ABB RobotStudio station: parte 2 - Lisandro y Camila.rspag

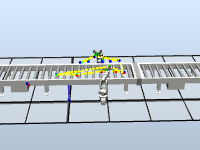
--- station ---
Station PARCIAL_FINAL_20 (saved by RobotStudio 6.8.8307.1040)
Controller IRB_120_3kg_0.58m_izqueirdo, task T_ROB1: task frame (RAPID world) sits at (1975.54, -890.46, 0) mm, rotated rx 0 ry 0 rz 180 deg in the station
Controller IRB_120_3kg_0.58m, task T_ROB1: task frame (RAPID world) sits at (-16.49, -890.46, 0) mm in the station
Controller IRB_120_3kg_0.58m
  mechanical unit ROB_1: IRB120_derecho, 6 joints, base frame (0, 0, 0) mm
Controller IRB_120_3kg_0.58m_izqueirdo
  mechanical unit ROB_1: IRB120_izquierdo, 6 joints, base frame (0, 0, 0) mm
Layout (positions relative to the parent item):
  - IRB120_derecho [mechanism] at (-16.49, -890.46, 0) mm; joint values [-0.3384, 0.2785, -0.49, -0.1645, -0.0408, 0.5646] (rad or m)
      links: Base, Link1, Link2, Link3, Link4, Link5, Link6
  - MyTool_derecho [mechanism] at (384.12, -1030.96, 699.37) mm, rotated rx 56.47 ry 63.2 rz 40.4 deg
      TCP MyTool at (31.79, 0, 229.64) mm, rotated rx 0 ry 38 rz 0 deg
      links: SpintecTool
  - SmartComponent_1 [smart component]
      signals: DI INICIO, DO DONE_1, DO WAIT_ROBOT, DI WAIT_ROBOT_1
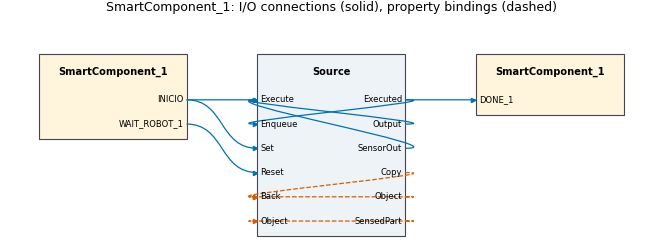
      connections:
        SmartComponent_1.INICIO -> Source.Execute
        Source.Executed -> Queue.Enqueue
        LogicSRLatch_2.Output -> LinearMover.Execute
        SmartComponent_1.INICIO -> LogicSRLatch_2.Set
        LineSensor.SensorOut -> Sink.Execute
        Sink.Executed -> SmartComponent_1.DONE_1
        SmartComponent_1.WAIT_ROBOT_1 -> LogicSRLatch_2.Reset
        Source.Copy => Queue.Back
        LinearMover.Object => Queue.Back
        LineSensor.SensedPart => Sink.Object
    - 950_4000_h2 [part] at (481.84, -1943.26, 0) mm, rotated rx 0 ry 0 rz -90 deg
    - 950_4000 [part] at (481.84, 2303.05, 0) mm, rotated rx 0 ry 0 rz -90 deg
  - LineSensor_3 [smart component, from Components\LineSensor.rslib] at (0, 0, 82.21) mm
      properties: Start=[0.481837 -1.468577 0.417790711533662]; End=[1.391837 -1.454228 0.417790711533662]; Radius=0; SensedPart=(none); SensedPoint=[1.1188828125 -1.45853198242187 0.5]
    - _sensorPart_ [part]
  - LinearMover_5 [smart component, from Components\LinearMover.rslib]
      properties: Object=(none); Direction=[0 -5 0]; Speed=0.45; Reference=Global; ReferenceObject=(none)
  - LogicSRLatch_3 [smart component, from Components\LogicSRLatch.rslib]
  - carro v10_9 [part] at (845.35, 1324.55, 563.17) mm, rotated rx 90 ry 0 rz 90 deg
  - Queue [smart component, from Components\Queue.rslib]
      properties: Back=(none); Front=(none); Queue={2e9f6991-8765-46e1-b9d2-2ffc72d677af};{ae45a596-02e8-4e52-9286-656ae225cacd};{e6612efd-c0eb-488b-85f8-b7f4c3102223};{41649e3c-b784-4099-a2b6-5bbce63e6931};{7cccd143-9200-41c9-9571-56f89e3b47af};{9ae8a6fd-c274-4031-a548-9f3ef3f36b3a};{8e4b5e29-5d32-45ba-96b5-431f4aa4aeb4};{b12dc332-1d97-4a47-8d88-8e0bee83711f};{b06eb078-9d15-4dac-a639-ca4a5d045752};{36dd95e1-a525-41dc-89b9-a063a131a275};{90e40d64-8709-426d-9514-00f99289b4fd};{8238a00f-e375-4470-8a06-12bd71f22f04};{9cebabc8-3cf8-4b9a-aff2-1a40ba7d75c4};{e08df943-d758-42c3-b96e-c5a5a5535acf};{779e000a-15d6-42ef-9bae-f04b49e1bf69};{19063376-c3c8-401e-bc56-325a5b5330d4};{6fb3a925-9c96-444a-9cf6-2b48ab2bb77b};{b99dccf3-a9df-44c4-8768-e74e9a577921};{d042e8a6-24ab-4afd-8b08-62ef72f8d954};{469562c5-238e-4f1a-8a6a-e243ac061d49};{98599022-264f-40f7-abfe-657128622a59};{93bca168-39dd-414b-b794-00b031783849};{70e5a896-b097-490d-8be8-28998b22b420};{5813b6a1-ddc2-47c4-ac52-396df1c672e9};{180ec9fe-a73e-4834-8773-2bd90c542f4d};{68088890-b0b0-44d4-a72b-623dbc1f9591};{e385e6d6-b519-43fc-8129-9058077c405e};{fb7d959f-a590-4f16-a74b-a7969766d88b};{d415407e-bbc8-41df-8733-1a202f62ccfb};{3bfff912-d452-4fed-8fb6-201deedca72a};{e2d4b341-78bb-44fa-a800-ceced0670a4f};{baedb794-50eb-4695-9b41-42448fe955b1};{10d86464-9892-4255-8e29-7578ef2925c7};{514a4022-64fc-47d2-bc88-f3ff3a7435df};{87afceb3-19d2-40d5-b81b-794861be6da1};{30505d37-60bd-4412-8ca7-5a9feadde122};{d50750b3-7fed-419f-9bb7-134f78306727};{72818c27-da5f-4208-8d82-50bde2b66c7d}; NumberOfObjects=1
  - Sink [smart component, from Components\Sink.rslib]
      properties: Object=(none)
  - Source [smart component, from Components\Source.rslib]
      properties: Source=carro v10_9; Copy=(none); Parent=(none); Position=[0.84535 1.32455 0.56317]; Orientation=[1.5707963267949 0 1.5707963267949]; Transient=false; PhysicsBehavior=2
  - LinearMover_6 [smart component, from Components\LinearMover.rslib]
      properties: Object=(none); Direction=[0 -6 0]; Speed=0.45; Reference=Global; ReferenceObject=(none)
  - LogicSRLatch_4 [smart component, from Components\LogicSRLatch.rslib]
  - LineSensor_4 [smart component, from Components\LineSensor.rslib]
      properties: Start=[0.481837 -3.897492 0.5]; End=[1.391837 -3.903973 0.5]; Radius=0; SensedPart=(none); SensedPoint=[0 0 0]
    - _sensorPart_ [part]
  - MyTool_izquierdo [mechanism] at (1574.94, -749.96, 699.37) mm, rotated rx 56.47 ry 63.2 rz -139.6 deg
      TCP MyTool at (31.79, 0, 229.64) mm, rotated rx 0 ry 38 rz 0 deg
      links: SpintecTool
  - IRB120_izquierdo [mechanism] at (1975.54, -890.46, 0) mm, rotated rx 0 ry 0 rz 180 deg; joint values [-0.3384, 0.2785, -0.49, -0.1645, -0.0408, 0.5645] (rad or m)
      links: Base, Link1, Link2, Link3, Link4, Link5, Link6
Attachment: MyTool_derecho is attached to IRB120_derecho / Link6
Attachment: MyTool_izquierdo is attached to IRB120_izquierdo / Link6
Station signals: DI STAR_JOB, DI RESET_CARRITO, DO END
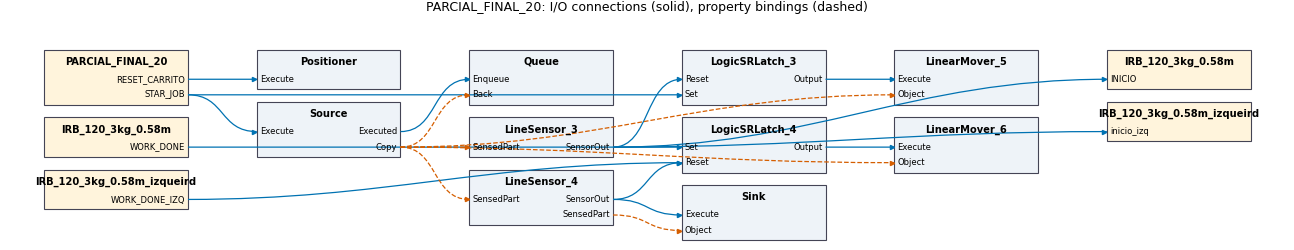
Station logic (signal -> signal, property => property):
  LineSensor_3.SensorOut -> LogicSRLatch_3.Reset
  LogicSRLatch_3.Output -> LinearMover_5.Execute
  PARCIAL_FINAL_20.RESET_CARRITO -> Positioner.Execute
  PARCIAL_FINAL_20.STAR_JOB -> Source.Execute
  Source.Executed -> Queue.Enqueue
  PARCIAL_FINAL_20.STAR_JOB -> LogicSRLatch_3.Set
  LineSensor_4.SensorOut -> Sink.Execute
  IRB_120_3kg_0.58m.WORK_DONE -> LogicSRLatch_4.Set
  LogicSRLatch_4.Output -> LinearMover_6.Execute
  LineSensor_4.SensorOut -> LogicSRLatch_4.Reset
  LineSensor_3.SensorOut -> IRB_120_3kg_0.58m.INICIO
  LineSensor_3.SensorOut -> IRB_120_3kg_0.58m_izqueirdo.inicio_izq
  IRB_120_3kg_0.58m_izqueirdo.WORK_DONE_IZQ -> LogicSRLatch_4.Reset
  Source.Copy => Queue.Back
  Source.Copy => LinearMover_5.Object
  Source.Copy => LinearMover_6.Object
  Source.Copy => LineSensor_4.SensedPart
  LineSensor_4.SensedPart => Sink.Object
  Source.Copy => LineSensor_3.SensedPart

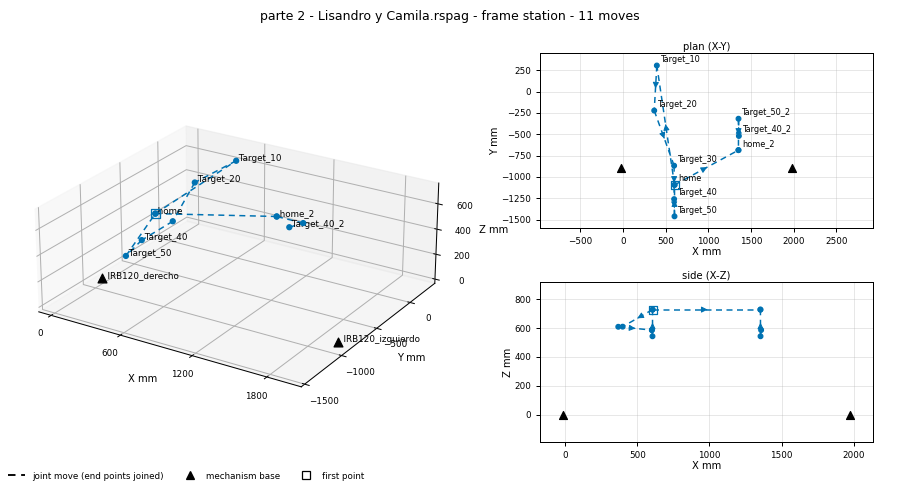
[picture p0: tool path of parte 2 - Lisandro y Camila.rspag in frame station, 11 of 14 moves have a stored position in this frame; points joined in program order, loops and branches not executed]
--- Backups/IRB_120_3kg_0.58m/RAPID/TASK1/PROGMOD/CalibData.mod ---
MODULE CalibData
	PERS tooldata MyTool;
	TASK PERS wobjdata Workobject_1:=[FALSE,TRUE,"",[[414.337,2008.173,310],[0.707106781,0,0,-0.707106781]],[[0,0,0],[1,0,0,0]]];
ENDMODULE

--- Backups/IRB_120_3kg_0.58m/RAPID/TASK1/PROGMOD/Module1.mod ---
MODULE Module1
	CONST robtarget Target_9:=[[1231.234317602,188.10759573,470.029292406],[0.397821209,-0.619255451,0.367382539,0.568586882],[0,-1,0,1],[9E+09,9E+09,9E+09,9E+09,9E+09,9E+09]];
	CONST robtarget Target_10:=[[813.404562568,-0.130130403,299.738578065],[0.271216707,-0.707758221,0.241098944,0.606127955],[0,0,-1,1],[9E+09,9E+09,9E+09,9E+09,9E+09,9E+09]];
	CONST robtarget Target_20:=[[1340.934,-30.557,299],[0.326505576,-0.627211375,0.627211375,0.326505576],[0,-2,1,0],[9E+09,9E+09,9E+09,9E+09,9E+09,9E+09]];
	CONST robtarget Target_30:=[[1986.491,202.361,276.17],[0.183012702,-0.683012702,0.683012702,0.183012702],[0,0,-1,0],[9E+09,9E+09,9E+09,9E+09,9E+09,9E+09]];
    CONST robtarget home:=[[2211.7760355,207.470989882,418.189910086],[0.328259674,-0.424354677,0.704665747,0.464343493],[-1,-1,-1,1],[9E+09,9E+09,9E+09,9E+09,9E+09,9E+09]];
    CONST robtarget Target_40:=[[2378.039,202.641,276.17],[0.271653782,-0.582563416,0.694272044,0.323744371],[0,-1,0,0],[9E+09,9E+09,9E+09,9E+09,9E+09,9E+09]];
    CONST robtarget Target_50:=[[2579.973,206.801,233.088],[0.64201571,-0.398058358,0.654107559,-0.038841622],[-1,-1,-1,1],[9E+09,9E+09,9E+09,9E+09,9E+09,9E+09]];
    !***********************************************************
    !
    ! Module:  Module1
    !
    ! Description:
    !   <Insert description here>
    !
    ! Author: camila
    !
    ! Version: 1.0
    !
    !***********************************************************


    !***********************************************************
    !
    ! Procedure main
    !
    !   This is the entry point of your program
    !
    !***********************************************************
    PROC main()
        !Add your code here
    ENDPROC
	PROC Path_10()
        WaitDI INICIO,1;
        MoveJ home,v500,fine,MyTool\WObj:=Workobject_1;
        MoveJ Target_10,v500,fine,MyTool\WObj:=Workobject_1;
        MoveJ Target_20,v500,fine,MyTool\WObj:=Workobject_1;
        MoveJ Target_30,v500,fine,MyTool\WObj:=Workobject_1;
        MoveJ Target_40,v500,fine,MyTool\WObj:=Workobject_1;
        MoveJ Target_50,v500,fine,MyTool\WObj:=Workobject_1;
        MoveJ home,v500,fine,MyTool\WObj:=Workobject_1;
        SetDO WORK_DONE,1;
	ENDPROC
ENDMODULE

--- Backups/IRB_120_3kg_0.58m_izqueirdo/RAPID/TASK1/PROGMOD/CalibData.mod ---
MODULE CalibData
	PERS tooldata MyTool:=[TRUE,[[31.792631019,0,229.638935148],[0.945518576,0,0.325568154,0]],[1,[0,0,1],[1,0,0,0],0,0,0]];
	TASK PERS wobjdata Workobject_1:=[FALSE,TRUE,"",[[414.337,2008.173,310],[0.707106781,0,0,-0.707106781]],[[0,0,0],[1,0,0,0]]];
	TASK PERS wobjdata Workobject_IZQ:=[FALSE,TRUE,"",[[414.337,2008.173,310],[0.707106781,0,0,-0.707106781]],[[0,0,0],[1,0,0,0]]];
ENDMODULE

--- Backups/IRB_120_3kg_0.58m_izqueirdo/RAPID/TASK1/PROGMOD/Module1.mod ---
MODULE Module1
	CONST robtarget home_2:=[[2211.7760355,207.470989882,418.189910086],[0.328259674,-0.424354677,0.704665747,0.464343493],[-1,-1,-1,1],[9E+09,9E+09,9E+09,9E+09,9E+09,9E+09]];
	CONST robtarget Target_30_2:=[[1986.491,202.361,276.17],[0.183012702,-0.683012702,0.683012702,0.183012702],[0,0,-1,0],[9E+09,9E+09,9E+09,9E+09,9E+09,9E+09]];
	CONST robtarget Target_40_2:=[[2378.039,202.641,276.17],[0.271653782,-0.582563416,0.694272044,0.323744371],[0,-1,0,0],[9E+09,9E+09,9E+09,9E+09,9E+09,9E+09]];
	CONST robtarget Target_50_2:=[[2579.973,206.801,233.088],[0.64201571,-0.398058358,0.654107559,-0.038841622],[-1,-1,-1,1],[9E+09,9E+09,9E+09,9E+09,9E+09,9E+09]];
	PROC Path_10()
	    WaitDI inicio_izq,1;
	    MoveJ home_2,v1000,z100,MyTool\WObj:=Workobject_IZQ;
	    MoveJ Target_10_2,v500,fine,MyTool\WObj:=Workobject_IZQ;
        MoveJ Target_20_2,v500,fine,MyTool\WObj:=Workobject_IZQ;
	    MoveJ Target__30_2,v500,fine,MyTool\WObj:=Workobject_IZQ;
	    MoveJ Target_40_2,v500,fine,MyTool\WObj:=Workobject_IZQ;
	    MoveJ Target_50_2,v500,fine,MyTool\WObj:=Workobject_IZQ;
	    MoveJ home_2,v500,fine,MyTool\WObj:=Workobject_IZQ;
	    SetDO WORK_DONE_IZQ,1;
	ENDPROC
ENDMODUL

--- Backups/IRB_120_3kg_0.58m/SYSPAR/EIO.cfg ---
EIO:CFG_1.0:6:1::
#
INDUSTRIAL_NETWORK:

      -Name "DeviceNet" -Label "DeviceNet Master/Slave Network" -Address "2"
#
DEVICENET_DEVICE:

      -Name "d652" -VendorName "ABB Robotics" -ProductName "24 VDC I/O Device"\
      -Label "DSQC 652 24 VDC I/O Device" -ProductCode 26 -DeviceType 7\
      -ConnectionType "COS" -OutputSize 2 -InputSize 2
#
DEVICENET_INTERNAL_DEVICE:

      -Name "DN_Internal_Device" -VendorName "ABB Robotics"\
      -ProductName "DeviceNet Internal Slave Device"
#
EIO_SIGNAL:

      -Name "WAIT_ROBOT" -SignalType "DO"

      -Name "INICIO" -SignalType "DI"

      -Name "WORK_DONE" -SignalType "DO"

      -Name "WAIT_TO_THE_END" -SignalType "DI"

--- Backups/IRB_120_3kg_0.58m_izqueirdo/SYSPAR/EIO.cfg ---
EIO:CFG_1.0:6:1::
#
INDUSTRIAL_NETWORK:

      -Name "DeviceNet" -Label "DeviceNet Master/Slave Network" -Address "2"
#
DEVICENET_INTERNAL_DEVICE:

      -Name "DN_Internal_Device" -VendorName "ABB Robotics"\
      -ProductName "DeviceNet Internal Slave Device"
#
EIO_SIGNAL:

      -Name "inicio_izq" -SignalType "DI"

      -Name "WAIT_ROBOT_IZQ" -SignalType "DO"

      -Name "WORK_DONE_IZQ" -SignalType "DO"
